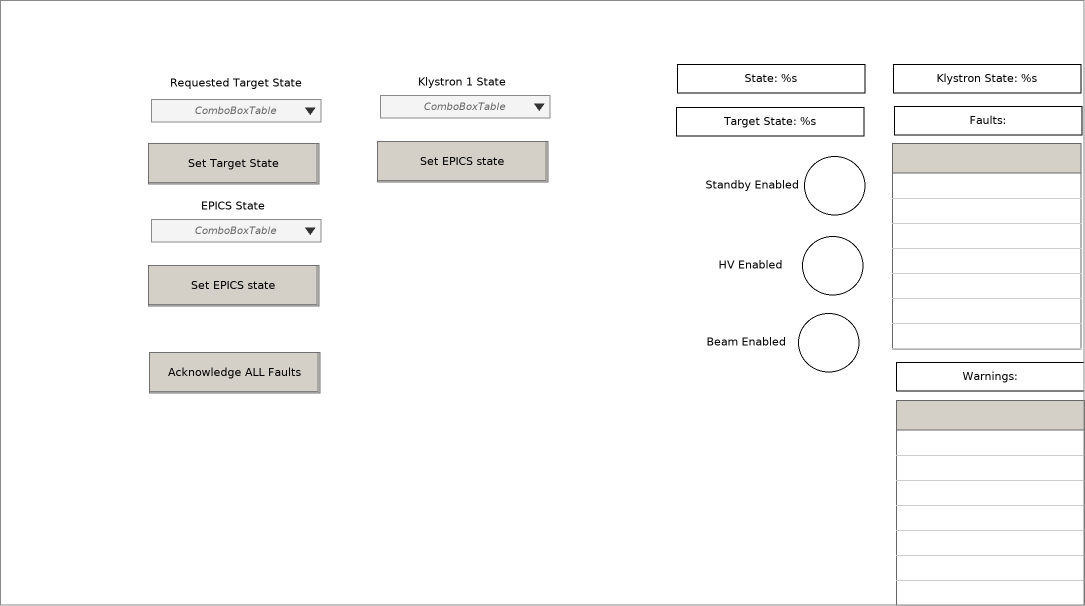
VISUALIZATION TestGUI  // 1085x606
    Button (148,143 171x41), "Set Target State"
        toggle MAIN.MpsLogicTest.SetTargetStateEPICS
    ComboBoxTable (151,99 170x23), variable: MAIN.MpsLogicTest.MpsSelectedTargetState, data array: MAIN.MpsLogicTest.MpsStateList
        p3854506369: MAIN.MpsLogicTest.MpsStateList[INDEX]
    Rectangle (677,64 188x29), "State: %s", text variable: MAIN.MpsLogicTest.StateController.State
    Ellipse (804,156 61x59), colour toggle: MAIN.MpsLogicTest.StandbyEnabled
    Label (703,170 99x30), "Standby Enabled"
    Ellipse (802,236 61x59), colour toggle: MAIN.MpsLogicTest.HVEnabled
    Label (701,250 99x30), "HV Enabled"
    Ellipse (798,313 61x59), colour toggle: MAIN.MpsLogicTest.BeamEnabled
    Label (697,327 99x30), "Beam Enabled"
    Rectangle (676,107 188x29), "Target State: %s", text variable: MAIN.MpsLogicTest.StateController.TargetState
    Rectangle (893,64 188x29), "Klystron State: %s", text variable: MAIN.MpsLogicTest.StateController.Klystron01State_RB
    Label (152,68 168x30), "Requested Target State"
    ComboBoxTable (151,219 170x23), variable: MAIN.MpsLogicTest.MpsSelectedEPICSState, data array: MAIN.MpsLogicTest.MpsStateList
        p3854506369: MAIN.MpsLogicTest.MpsStateList[INDEX]
    Label (148,191 170x30), "EPICS State"
    Button (148,265 171x41), "Set EPICS state"
        toggle MAIN.MpsLogicTest.SetEPICSState
    Table (892,143 189x206), data array: MAIN.MpsLogicTest.StateController.Fault_OUT
        p3854506369: MAIN.MpsLogicTest.StateController.Fault_OUT[INDEX]
        p2232123230: MAIN.MpsLogicTest.StateController.Fault[INDEX]
        p2685023577: MAIN.MpsLogicTest.StateController.Fault_OUT_OUT[INDEX]
    Table (896,400 189x206), data array: MAIN.MpsLogicTest.StateController.Warning_OUT
        p3854506369: MAIN.MpsLogicTest.StateController.Warning_OUT[INDEX]
        p2232123230: MAIN.MpsLogicTest.StateController.Warning[INDEX]
        p2685023577: MAIN.MpsLogicTest.StateController.Warning_OUT_OUT[INDEX]
    Rectangle (894,106 188x29), "Faults:"
    Rectangle (896,362 188x29), "Warnings:"
    Button (149,352 171x41), "Acknowledge ALL Faults"
        toggle G_Epics.General.AcknowledgeAllCmd
    ComboBoxTable (380,95 170x23), variable: MAIN.MpsLogicTest.StateController.Klystron01State_RB, data array: MAIN.MpsLogicTest.MpsStateList
        p3854506369: MAIN.MpsLogicTest.MpsStateList[INDEX]
    Label (377,67 170x30), "Klystron 1 State"
    Button (377,141 171x41), "Set EPICS state"
        toggle MAIN.MpsLogicTest.SetEPICSState
END_VISUALIZATION

(* stored: Version 1.1.0.1, ProductVersion 3.1.4024.12
   Visu TestGUI: Id {054b4fb3-dc26-4030-a3b4-5363aab83aa2} *)
